(* CoDeSys 2.3 export: ESTACION.EXP *)

(* Data type *)
TYPE Estacion :
STRUCT
	Cilindro_A  	          : Cilindro_Simple;
	Empty        			   : Sensor_Foto;
	Base_en_Posicion : Sensor_Cap;
END_STRUCT
END_TYPE
